FUNCTION_BLOCK ExecuteProduct (* JADE WORKER *)
  (* Standard: 61499-1 *)
  (* Version 1.0, 2014-04-22, Ahmed, Fraunhofer IGD *)
  (* Compiler header: package fb.rt; *)
  (* Compiler Java Sun JDK 1.5.0 *)
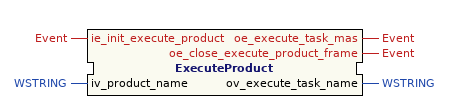
  EVENT_INPUT
    ie_init_execute_product;
  END_EVENT
  EVENT_OUTPUT
    oe_execute_task_mas;
    oe_close_execute_product_frame;
  END_EVENT
  VAR_INPUT
    iv_product_name : WSTRING;
  END_VAR
  VAR_OUTPUT
    ov_execute_task_name : WSTRING;
  END_VAR
END_FUNCTION_BLOCK
